TEXTLIST User
  0 = 'None'
  1 = 'Engineer'
  2 = 'Technician'
  3 = 'Operator'
   = ''
END_TEXTLIST

(* stored: Version 1.1.0.1, ProductVersion 3.1.4024.12
   TextList User: Id {fdd893b0-2ac7-4b72-9aa5-4486005a7963} *)
